{attribute clr [Container(Layout.Stack)]}
{attribute clr [Group(Layout.Scroll)]}
TYPE CUTechnologicalDataBase EXTENDS TcoCore.TcoStruct :
STRUCT
	{attribute wpf [Container(Layout.Stack,"General")]}
	{attribute wpf [Group(Layout.GroupBox)]}
	{attribute addProperty Name "<#Cycle time#> - <#Nominal#>"}
	IdealCycleTime   : TIME;
	
	{attribute addProperty Name "<#Cycle time#> - <#Warning#>"}
	WarningCycleTime : TIME;
    
	{attribute addProperty Name "<#Cycle time#> - <#Error#>"}
	ErrorCycleTime   : TIME;

	
	{attribute addProperty Name "<#Step time#> - <#Warning#>"}
	WarningStepAlarmTime : TIME;
    
	{attribute addProperty Name "<#Step time#> - <#Error#>"}
	ErrorStepAlarmTime   : TIME;
	
	{attribute addProperty Name "<#Energy saving mode - Inactivity time#> "}
	TimeToEntryEnergySavingMode : TIME;
	
	{attribute addProperty Name "<#No of allowed any recurring failures in seqence#> "}
	AnyRecurringFailure   : UINT;
	
	{attribute addProperty Name "<#No of allowed same recurring failures in seqence#> "}
	SameRecurringFailure   : UINT;
	
	
END_STRUCT
END_TYPE

(* stored: Version 1.1.0.1
   DUT CUTechnologicalDataBase: Id {7f1b525b-56fa-09a1-1f2d-f6d3ae7fbaf7} *)
